FUNCTION_BLOCK OpenCloseGarage
VAR_INPUT
	bActuationProgram : BOOL; //the input we give through the interfac
	bError : BOOL; //light that paused the door
END_VAR
VAR_OUTPUT
	bLight : BOOL; //garage light that turns on if the garage is opening or closing (blinks if there is an error or the garage failed to open/close
	bDoorOpen : BOOL; //sensor that indicates wheather or not the garage door is opened
	bDoorClosed : BOOL; //sensor that indicate wheather or not the garage is closed
	bDriveOverload : BOOL; //sensor that indicates if there is an error or if the garage takes too log to open/closLight
	bLightForPause : BOOL;
	bVisualization : BOOL; //bool varable for visual effects
END_VAR
VAR
	iState : UDINT; //states variable which we use to go through states
	fbOpen : TON; //time that opens the door
	fbClose : TON; //timer that closes the door
	fbInitial : R_TRIG; //trigger for setting the initial position of the door to closed
	bInitialActivate : BOOL; //bool variable that activates the initial trigger
	fbBlink : Blinker;
	bActuation : BOOL; //actuation button which closes/opens the door
	
	bTempOp : BOOL; //temp open variable, helps in the error state
	bTempCls : BOOL; //temp closed variable,helps in the error state
	
	fbActivate : R_TRIG; // trigger for activation
END_VAR

bInitialActivate := TRUE; //we close the door at the start
fbInitial(CLK := TRUE);
IF fbInitial.Q THEN
	bDoorClosed := TRUE; //we have set the door to closed at the start (only activates the first time we run the program
END_IF

CASE iState OF
	0:
		fbActivate(CLK := bActuationProgram);
		IF fbActivate.Q THEN
			bActuation := TRUE;
		END_IF
		IF bActuation THEN
			iState := 10; //if we click the button go to the next state and check it's state
		END_IF
	5: //forgot to turn off actuation added an extra state
		bActuation := FALSE;
		iState := 0; //return to the first state	
	10:
		IF bDoorOpen THEN
			bDoorOpen := FALSE;
			iState := 20; //if opened go to state 20
		ELSIF bDoorClosed THEN
			bDoorClosed := FALSE;
			iState := 30; //if closed go to state 30
		ELSIF bDriveOverload THEN
			bDoorClosed := FALSE;
			bDoorOpen := FALSE;
			bActuation := FALSE; //we turn off the actuation button
			iState := 50; //if there is an error go to state 40
		END_IF
	15:
		bActuation := FALSE;
		iState := 50;
	20:	
		fbActivate(CLK := bActuationProgram);
		IF fbActivate.Q THEN
			bActuation := FALSE;
		END_IF	
		IF bError THEN
			iState := 15; //incase the door goes to error
		END_IF
		IF bActuation THEN
			fbClose.IN := TRUE; //we start closing it
			bLight := TRUE; //we turn the light on             
			bTempCls := TRUE; //set the temp to true
			IF fbClose.Q THEN //if it finished closing
				bTempCls := FALSE; //set the temp to false
				bDoorClosed := TRUE; //turn the closed sensor on
				fbClose.IN := FALSE; //reset timer
				bLight := FALSE; //turn the light off
				iState := 5; //turn off actuation
			END_IF
		ELSE
			bLightForPause := TRUE;
			iState := 40; //if we stopped the door go to the pause state
		END_IF

			
	30: //if the door is closed
		fbActivate(CLK := bActuationProgram);
		IF fbActivate.Q THEN
			bActuation := FALSE;
		END_IF
		IF bError THEN
			iState := 15; //incase the door goes to error
		END_IF
		IF bActuation THEN
			fbOpen.IN := TRUE; //we start opening it
			bLight := TRUE; //we turn the light on
			bTempOp := TRUE;// set the temp open to true
			IF fbOpen.Q THEN //if it finished opening
				bTempOp := FALSE;
				bDoorOpen := TRUE; //turn the open sensor on
				fbOpen.IN := FALSE; //reset timer
				bLight := FALSE; //turn the light off
				iState := 5; //turn off actuation
			END_IF
		ELSE
			bLightForPause := TRUE;
			iState := 40; //if we paused the door go to the pause state for open
		END_IF
	40:
		IF bError THEN
			bDriveOverload := TRUE;
			iState := 15; //incase the door goes to error
		END_IF
		bVisualization := TRUE;
		fbOpen.IN := FALSE; //reset the timers
		fbClose.IN := FALSE;
		bDoorClosed := FALSE;
		bDoorOpen := FALSE; //we set the door states to false
		fbActivate(CLK := bActuationProgram);
		IF fbActivate.Q THEN
			bActuation := TRUE;
			bLightForPause := FALSE; //we turn off the pause light
		END_IF
		IF bActuation AND bTempOp THEN //if we press the actuation button and the door was opening
			bLight := TRUE;
			fbClose.IN := TRUE;
			IF fbClose.Q THEN
				bVisualization := FALSE;
				bDoorClosed := TRUE; //we closed the door
 				bLight := FALSE;
				bTempOp := FALSE;
				fbClose.IN := FALSE;
				bDriveOverload := FALSE;
				iState := 5; //turn off actuation
			END_IF	
		END_IF
		IF bActuation AND bTempCls THEN //if we press the actuation button and the door was opening
			bLight := TRUE;
			fbOpen.IN := TRUE;
			IF fbOpen.Q THEN
				bVisualization := FALSE;
				bDoorOpen := TRUE; //we opened the door
 				bLight := FALSE;
				bTempCls := FALSE;
				fbOpen.IN := FALSE;
				bDriveOverload := FALSE;
				iState := 5; //turn actuation off
			END_IF	
		END_IF
				
	50: //error state
		bLight := fbBlink.bBlink; //we mak the light blink
		fbBlink();
		bDriveOverload := TRUE;
		fbOpen.IN := FALSE; //reset the timers
		fbClose.IN := FALSE;
		bDoorClosed := FALSE;
		bDoorOpen := FALSE; //we set the door states to false
		bVisualization := FALSE;
		bLightForPause := FALSE;
		fbActivate(CLK := bActuationProgram);
		IF fbActivate.Q THEN
			bActuation := TRUE;
		END_IF
		IF bActuation AND bTempOp THEN //if we press the actuation button and the door was opening
			bLight := TRUE;
			fbClose.IN := TRUE;
			bDriveOverload := FALSE;
			IF fbClose.Q THEN
				bDoorClosed := TRUE; //we closed the door
 				bLight := FALSE;
				bTempOp := FALSE;
				fbClose.IN := FALSE;
				iState := 5; //turn off actuation
			END_IF	
		END_IF
		IF bActuation AND bTempCls THEN //if we press the actuation button and the door was opening
			bLight := TRUE;
			fbOpen.IN := TRUE;
			bDriveOverload := FALSE;
			IF fbOpen.Q THEN
				bDoorOpen := TRUE; //we opened the door
 				bLight := FALSE;
				bTempCls := FALSE;
				fbOpen.IN := FALSE;
				iState := 5; //turn actuation off
			END_IF	
		END_IF
END_CASE

fbOpen(PT := T#7000MS);
fbClose(PT := T#7000MS);

END_FUNCTION_BLOCK

(* stored: Version 1.1.0.1, ProductVersion 3.1.4024.12
   POU OpenCloseGarage: Id {729de886-c8a7-444c-9b8a-a55b37bcaac6}, SpecialFunc None *)
